FUNCTION_BLOCK EL1004
VAR
	_io : EL1xx4_Data;
	{attribute addProperty Name "WcState"}
	_wcState : WcStateInputToggle;
	{attribute addProperty Name "Info data"}
	_infoData : InfoDataBase;
END_VAR

PROPERTY IO : REFERENCE TO EL1xx4_Data
GET
IO REF= _io;
END_GET
END_PROPERTY

PROPERTY WcState : REFERENCE TO WcStateInputToggle
GET
WcState REF= _wcState;
END_GET
END_PROPERTY

END_FUNCTION_BLOCK

(* stored: Version 1.1.0.1, ProductVersion 3.1.4024.9
   POU EL1004: Id {3a867e3f-848e-0a24-13dc-fb4382521a0c}, SpecialFunc None
   Property IO: Id {4eddd268-92ab-0beb-2455-7becd4c61e10}
   Get Get: Id {e1caf375-d05d-0232-0990-545eab20bb86}
   Property WcState: Id {d84fc244-a475-06ea-0cf8-61eb6bcd4832}
   Get Get: Id {7e0980e6-fe3b-0e96-110e-fb750da443eb} *)
